(* Logix 5000 project; controller NSutherlandCapstone Emulate 5570 rev 32.11; software revision 32.00 *)

TASK MainTask (continuous, watchdog 500 ms) : MainProgram, _3WireControl, GarageDoor

MODULES
   Local : Emulate 5570 (ICP 0, rev 32.11)
      IO_Simulator : vendor 1 type 0 code 15 (ICP 3, rev 1.1, Output RPI 5 ms)
END_MODULES

VAR_GLOBAL   (* controller tags *)
   PL_G : BOOL := 1;
   PL_R : BOOL;
   SS : BOOL;
END_VAR

PROGRAM _3WireControl   (* main routine MainRoutine *)
// PLC lab 3
VAR
   Motor : BOOL;
   NCNC_AND_00 : FBD_BOOLEAN_AND := (In1 := 1, In2 := 1, In3 := 1, In4 := 1, In5 := 1, In6 := 1, In7 := 1, In8 := 1);
   NCNC_Motor_Energize : SFC_ACTION := (Status := 16#0020_0000, PauseTimer := 1);
   NCNC_NOT_00 : FBD_BOOLEAN_NOT := (In := 1);
   NCNC_OR_00 : FBD_BOOLEAN_OR;
   NCNC_SetBit : SFC_STEP := (Status := 16#0020_0000, PauseTimer := 1);
   NCNC_SetDone : BOOL;
   NCNO_AND_00 : FBD_BOOLEAN_AND := (In1 := 1, In2 := 1, In3 := 1, In4 := 1, In5 := 1, In6 := 1, In7 := 1, In8 := 1);
   NCNO_Motor_Energize : SFC_ACTION := (Status := 16#0020_0000, PauseTimer := 1);
   NCNO_OR_00 : FBD_BOOLEAN_OR;
   NCNO_SetBit : SFC_STEP := (Status := 16#0020_0000, PauseTimer := 1);
   NCNO_SetDone : BOOL;
   NONC_AND_00 : FBD_BOOLEAN_AND := (In1 := 1, In2 := 1, In3 := 1, In4 := 1, In5 := 1, In6 := 1, In7 := 1, In8 := 1);
   NONC_Motor_Energize : SFC_ACTION := (Status := 16#0020_0000, PauseTimer := 1);
   NONC_NOT_00 : FBD_BOOLEAN_NOT := (In := 1);
   NONC_NOT_01 : FBD_BOOLEAN_NOT := (In := 1);
   NONC_OR_00 : FBD_BOOLEAN_OR;
   NONC_SetBit : SFC_STEP := (Status := 16#0020_0000, PauseTimer := 1);
   NONC_SetDone : BOOL;
   NONO_AND_00 : FBD_BOOLEAN_AND := (In1 := 1, In2 := 1, In3 := 1, In4 := 1, In5 := 1, In6 := 1, In7 := 1, In8 := 1);
   NONO_Motor_Energize : SFC_ACTION := (Status := 16#0020_0000, PauseTimer := 1);
   NONO_NOT_00 : FBD_BOOLEAN_NOT := (In := 1);
   NONO_OR_00 : FBD_BOOLEAN_OR;
   NONO_SetBit : SFC_STEP := (Status := 16#0020_0000, PauseTimer := 1);
   NONO_SetDone : BOOL;
   PB1 : BOOL := 1;   // NC PB
   PB2 : BOOL;   // NO PB
   PB3 : BOOL;   // NO PB
   PB4 : BOOL := 1;   // NC PB
END_VAR

ROUTINE FBD_1_NCNO   (* function block diagram *)
   SHEET 1
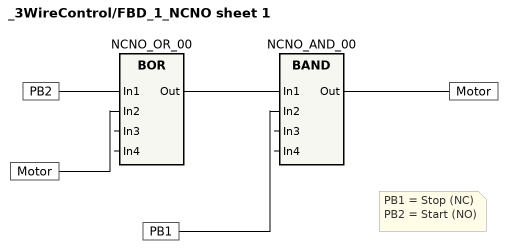
   // PB1 = Stop (NC)
   // PB2 = Start (NO)
   NCNO_OR_00 : BOR(In1 := PB2, In2 := Motor);   // unwired pins: In3 In4
   NCNO_AND_00 : BAND(In1 := NCNO_OR_00.Out, In2 := PB1);   // unwired pins: In3 In4
   Motor := NCNO_AND_00.Out;
END_ROUTINE

ROUTINE FBD_2_NONO   (* function block diagram *)
   SHEET 1
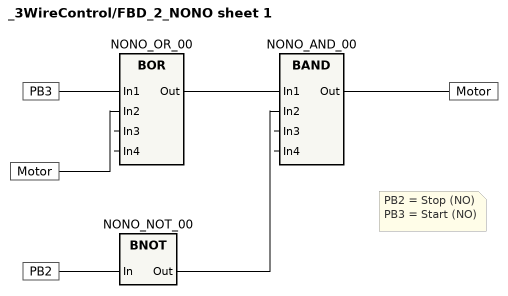
   // PB2 = Stop (NO)
   // PB3 = Start (NO)
   NONO_OR_00 : BOR(In1 := PB3, In2 := Motor);   // unwired pins: In3 In4
   NONO_NOT_00 : BNOT(In := PB2);
   NONO_AND_00 : BAND(In1 := NONO_OR_00.Out, In2 := NONO_NOT_00.Out);   // unwired pins: In3 In4
   Motor := NONO_AND_00.Out;
END_ROUTINE

ROUTINE FBD_3_NONC   (* function block diagram *)
   SHEET 1
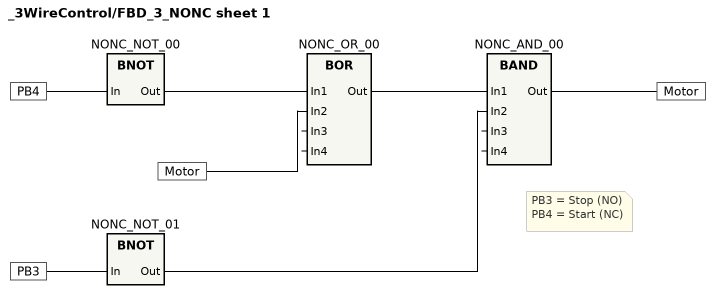
   // PB3 = Stop (NO)
   // PB4 = Start (NC)
   NONC_NOT_00 : BNOT(In := PB4);
   NONC_NOT_01 : BNOT(In := PB3);
   NONC_OR_00 : BOR(In1 := NONC_NOT_00.Out, In2 := Motor);   // unwired pins: In3 In4
   NONC_AND_00 : BAND(In1 := NONC_OR_00.Out, In2 := NONC_NOT_01.Out);   // unwired pins: In3 In4
   Motor := NONC_AND_00.Out;
END_ROUTINE

ROUTINE FBD_4_NCNC   (* function block diagram *)
   SHEET 1
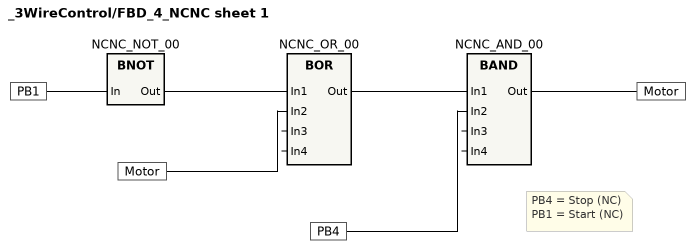
   // PB4 = Stop (NC)
   // PB1 = Start (NC)
   NCNC_NOT_00 : BNOT(In := PB1);
   NCNC_OR_00 : BOR(In1 := NCNC_NOT_00.Out, In2 := Motor);   // unwired pins: In3 In4
   NCNC_AND_00 : BAND(In1 := NCNC_OR_00.Out, In2 := PB4);   // unwired pins: In3 In4
   Motor := NCNC_AND_00.Out;
END_ROUTINE

ROUTINE MainRoutine   (* structured text *)
   JSR(SFC_3_NONC);
END_ROUTINE

ROUTINE SFC_1_NCNO   (* sequential function chart *)
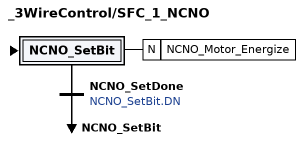
   INITIAL_STEP NCNO_SetBit:
      ACTION NCNO_Motor_Energize (N):
         Motor := PB1 & (PB2 OR Motor);
      END_ACTION
   END_STEP
   TRANSITION NCNO_SetDone FROM NCNO_SetBit TO NCNO_SetBit
      := NCNO_SetBit.DN
   END_TRANSITION
END_ROUTINE

ROUTINE SFC_2_NONO   (* sequential function chart *)
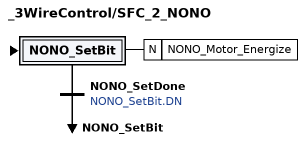
   INITIAL_STEP NONO_SetBit:
      ACTION NONO_Motor_Energize (N):
         Motor := NOT PB2 & (PB3 OR Motor);
      END_ACTION
   END_STEP
   TRANSITION NONO_SetDone FROM NONO_SetBit TO NONO_SetBit
      := NONO_SetBit.DN
   END_TRANSITION
END_ROUTINE

ROUTINE SFC_3_NONC   (* sequential function chart *)
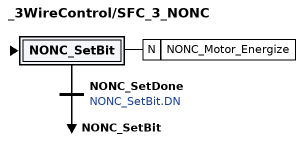
   INITIAL_STEP NONC_SetBit:
      ACTION NONC_Motor_Energize (N):
         Motor := NOT PB3 & (NOT PB4 OR Motor);
      END_ACTION
   END_STEP
   TRANSITION NONC_SetDone FROM NONC_SetBit TO NONC_SetBit
      := NONC_SetBit.DN
   END_TRANSITION
END_ROUTINE

ROUTINE SFC_4_NCNC   (* sequential function chart *)
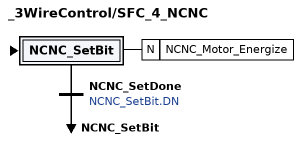
   INITIAL_STEP NCNC_SetBit:
      ACTION NCNC_Motor_Energize (N):
         Motor := PB4 & (NOT PB1 OR Motor);
      END_ACTION
   END_STEP
   TRANSITION NCNC_SetDone FROM NCNC_SetBit TO NCNC_SetBit
      := NCNC_SetBit.DN
   END_TRANSITION
END_ROUTINE

ROUTINE ST_1_NCNO   (* structured text *)
// Routine 1 of PLC lab 3
   // Lab 3 R1_NCNO
   (*
       PB1 = NC PB
       PB2 = NO PB
   *)
   
   Motor := PB1 & (PB2 OR Motor);
END_ROUTINE

ROUTINE ST_2_NONO   (* structured text *)
// Routine 2 of PLC lab 3
   // Lab 3 R2_NONO
   (*
       PB3 = NO PB
       PB2 = NO PB
   *)
   
   Motor := NOT PB2 & (PB3 OR Motor);
END_ROUTINE

ROUTINE ST_3_NONC   (* structured text *)
// Routine 3 of PLC lab 3
   // Lab 3 R3_NONC
   (*
       PB3 = NO PB
       PB4 = NC PB
   *)
   
   Motor := NOT PB3 & (NOT PB4 OR Motor);
END_ROUTINE

ROUTINE ST_4_NCNC   (* structured text *)
// Routine 4 of PLC lab 3
   // Lab 3 R4_NCNC
   (*
        PB4 = NC PB
        PB1 = NC PB
   *)
   
   Motor := PB4 & (NOT PB1 OR Motor);
END_ROUTINE
END_PROGRAM

PROGRAM GarageDoor   (* main routine MainRoutine *)
// PLC lab 4
VAR
   Ajar_LT : BOOL := 1;
   Bottom_Sensor : BOOL;
   Closed_LT : BOOL;
   Down_PB : BOOL;
   Fault_LT : BOOL;
   Halt : BOOL;
   Motor_Down : BOOL;
   Motor_Stopped : BOOL := 1;
   Motor_Up : BOOL;
   Open_LT : BOOL;
   Stop_PB : BOOL;
   Top_Sensor : BOOL;
   Up_PB : BOOL;
   Ver1_AND_00 : FBD_BOOLEAN_AND := (In1 := 1, In2 := 1, In3 := 1, In4 := 1, In5 := 1, In6 := 1, In7 := 1, In8 := 1);
   Ver1_AND_01 : FBD_BOOLEAN_AND := (In1 := 1, In2 := 1, In3 := 1, In4 := 1, In5 := 1, In6 := 1, In7 := 1, In8 := 1);
   Ver1_AND_02 : FBD_BOOLEAN_AND := (In1 := 1, In2 := 1, In3 := 1, In4 := 1, In5 := 1, In6 := 1, In7 := 1, In8 := 1);
   Ver1_AND_03 : FBD_BOOLEAN_AND := (In1 := 1, In2 := 1, In3 := 1, In4 := 1, In5 := 1, In6 := 1, In7 := 1, In8 := 1);
   Ver1_AND_04 : FBD_BOOLEAN_AND := (In1 := 1, In2 := 1, In3 := 1, In4 := 1, In5 := 1, In6 := 1, In7 := 1, In8 := 1);
   Ver1_AND_05 : FBD_BOOLEAN_AND := (In1 := 1, In2 := 1, In3 := 1, In4 := 1, In5 := 1, In6 := 1, In7 := 1, In8 := 1);
   Ver1_AND_06 : FBD_BOOLEAN_AND := (In1 := 1, In2 := 1, In3 := 1, In4 := 1, In5 := 1, In6 := 1, In7 := 1, In8 := 1);
   Ver1_AND_07 : FBD_BOOLEAN_AND := (In1 := 1, In2 := 1, In3 := 1, In4 := 1, In5 := 1, In6 := 1, In7 := 1, In8 := 1);
   Ver1_AND_08 : FBD_BOOLEAN_AND := (In1 := 1, In2 := 1, In3 := 1, In4 := 1, In5 := 1, In6 := 1, In7 := 1, In8 := 1);
   Ver1_MotorEnergize : SFC_ACTION := (Status := 16#0020_0000, PauseTimer := 1);
   Ver1_NOT_00 : FBD_BOOLEAN_NOT := (In := 1);
   Ver1_NOT_01 : FBD_BOOLEAN_NOT := (In := 1);
   Ver1_NOT_02 : FBD_BOOLEAN_NOT := (In := 1);
   Ver1_NOT_03 : FBD_BOOLEAN_NOT := (In := 1);
   Ver1_NOT_04 : FBD_BOOLEAN_NOT := (In := 1);
   Ver1_NOT_05 : FBD_BOOLEAN_NOT := (In := 1);
   Ver1_NOT_06 : FBD_BOOLEAN_NOT := (In := 1);
   Ver1_NOT_07 : FBD_BOOLEAN_NOT := (In := 1);
   Ver1_NOT_08 : FBD_BOOLEAN_NOT := (In := 1);
   Ver1_NOT_09 : FBD_BOOLEAN_NOT := (In := 1);
   Ver1_NOT_10 : FBD_BOOLEAN_NOT := (In := 1);
   Ver1_NOT_11 : FBD_BOOLEAN_NOT := (In := 1);
   Ver1_NOT_12 : FBD_BOOLEAN_NOT := (In := 1);
   Ver1_NOT_13 : FBD_BOOLEAN_NOT := (In := 1);
   Ver1_OR_00 : FBD_BOOLEAN_OR;
   Ver1_OR_01 : FBD_BOOLEAN_OR;
   Ver1_SetBit : SFC_STEP := (Status := 16#0020_0000, PauseTimer := 1);
   Ver1_SetDone : BOOL;
   Ver1_SetIndicators : SFC_ACTION := (Status := 16#0020_0000, PauseTimer := 1);
   Ver2_AND_00 : FBD_BOOLEAN_AND := (In1 := 1, In2 := 1, In3 := 1, In4 := 1, In5 := 1, In6 := 1, In7 := 1, In8 := 1);
   Ver2_AND_01 : FBD_BOOLEAN_AND := (In1 := 1, In2 := 1, In3 := 1, In4 := 1, In5 := 1, In6 := 1, In7 := 1, In8 := 1);
   Ver2_AND_02 : FBD_BOOLEAN_AND := (In1 := 1, In2 := 1, In3 := 1, In4 := 1, In5 := 1, In6 := 1, In7 := 1, In8 := 1);
   Ver2_AND_03 : FBD_BOOLEAN_AND := (In1 := 1, In2 := 1, In3 := 1, In4 := 1, In5 := 1, In6 := 1, In7 := 1, In8 := 1);
   Ver2_AND_04 : FBD_BOOLEAN_AND := (In1 := 1, In2 := 1, In3 := 1, In4 := 1, In5 := 1, In6 := 1, In7 := 1, In8 := 1);
   Ver2_AND_05 : FBD_BOOLEAN_AND := (In1 := 1, In2 := 1, In3 := 1, In4 := 1, In5 := 1, In6 := 1, In7 := 1, In8 := 1);
   Ver2_AND_06 : FBD_BOOLEAN_AND := (In1 := 1, In2 := 1, In3 := 1, In4 := 1, In5 := 1, In6 := 1, In7 := 1, In8 := 1);
   Ver2_AND_07 : FBD_BOOLEAN_AND := (In1 := 1, In2 := 1, In3 := 1, In4 := 1, In5 := 1, In6 := 1, In7 := 1, In8 := 1);
   Ver2_AND_08 : FBD_BOOLEAN_AND := (In1 := 1, In2 := 1, In3 := 1, In4 := 1, In5 := 1, In6 := 1, In7 := 1, In8 := 1);
   Ver2_AND_09 : FBD_BOOLEAN_AND := (In1 := 1, In2 := 1, In3 := 1, In4 := 1, In5 := 1, In6 := 1, In7 := 1, In8 := 1);
   Ver2_AND_10 : FBD_BOOLEAN_AND := (In1 := 1, In2 := 1, In3 := 1, In4 := 1, In5 := 1, In6 := 1, In7 := 1, In8 := 1);
   Ver2_AND_11 : FBD_BOOLEAN_AND := (In1 := 1, In2 := 1, In3 := 1, In4 := 1, In5 := 1, In6 := 1, In7 := 1, In8 := 1);
   Ver2_AND_12 : FBD_BOOLEAN_AND := (In1 := 1, In2 := 1, In3 := 1, In4 := 1, In5 := 1, In6 := 1, In7 := 1, In8 := 1);
   Ver2_CheckAjar : BOOL;
   Ver2_CheckClosed : BOOL;
   Ver2_CheckDown : BOOL;
   Ver2_CheckFault : BOOL;
   Ver2_CheckHalt : BOOL;
   Ver2_CheckOpen : BOOL;
   Ver2_CheckStopped : BOOL;
   Ver2_CheckUp : BOOL;
   Ver2_DoneAjar : BOOL;
   Ver2_DoneClosed : BOOL;
   Ver2_DoneDown : BOOL;
   Ver2_DoneFault : BOOL;
   Ver2_DoneHalt : BOOL;
   Ver2_DoneOpen : BOOL;
   Ver2_DoneStopped : BOOL;
   Ver2_DoneUp : BOOL;
   Ver2_MotorEnergize : SFC_ACTION := (Status := 16#0020_0000, PauseTimer := 1);
   Ver2_NOT_00 : FBD_BOOLEAN_NOT := (In := 1);
   Ver2_NOT_01 : FBD_BOOLEAN_NOT := (In := 1);
   Ver2_NOT_02 : FBD_BOOLEAN_NOT := (In := 1);
   Ver2_NOT_03 : FBD_BOOLEAN_NOT := (In := 1);
   Ver2_NOT_04 : FBD_BOOLEAN_NOT := (In := 1);
   Ver2_NOT_05 : FBD_BOOLEAN_NOT := (In := 1);
   Ver2_NOT_06 : FBD_BOOLEAN_NOT := (In := 1);
   Ver2_NOT_07 : FBD_BOOLEAN_NOT := (In := 1);
   Ver2_NOT_08 : FBD_BOOLEAN_NOT := (In := 1);
   Ver2_NOT_09 : FBD_BOOLEAN_NOT := (In := 1);
   Ver2_NOT_10 : FBD_BOOLEAN_NOT := (In := 1);
   Ver2_NOT_11 : FBD_BOOLEAN_NOT := (In := 1);
   Ver2_NOT_12 : FBD_BOOLEAN_NOT := (In := 1);
   Ver2_NOT_13 : FBD_BOOLEAN_NOT := (In := 1);
   Ver2_OR_00 : FBD_BOOLEAN_OR;
   Ver2_OR_01 : FBD_BOOLEAN_OR;
   Ver2_OR_02 : FBD_BOOLEAN_OR;
   Ver2_OR_03 : FBD_BOOLEAN_OR;
   Ver2_OR_04 : FBD_BOOLEAN_OR;
   Ver2_SetAjar : SFC_ACTION := (Status := 16#0020_0000, PauseTimer := 1);
   Ver2_SetBit : SFC_STEP := (Status := 16#0020_0000, PauseTimer := 1);
   Ver2_SetBit0 : SFC_STEP := (Status := 16#0020_0000, PauseTimer := 1);
   Ver2_SetBit1 : SFC_STEP := (Status := 16#0020_0000, PauseTimer := 1);
   Ver2_SetBit2 : SFC_STEP := (Status := 16#0020_0000, PauseTimer := 1);
   Ver2_SetBit3 : SFC_STEP := (Status := 16#0020_0000, PauseTimer := 1);
   Ver2_SetBit4 : SFC_STEP := (Status := 16#0020_0000, PauseTimer := 1);
   Ver2_SetBit5 : SFC_STEP := (Status := 16#0020_0000, PauseTimer := 1);
   Ver2_SetBit6 : SFC_STEP := (Status := 16#0020_0000, PauseTimer := 1);
   Ver2_SetBit7 : SFC_STEP := (Status := 16#0020_0000, PauseTimer := 1);
   Ver2_SetClosed : SFC_ACTION := (Status := 16#0020_0000, PauseTimer := 1);
   Ver2_SetDone : BOOL;
   Ver2_SetDown : SFC_ACTION := (Status := 16#0020_0000, PauseTimer := 1);
   Ver2_SetFault : SFC_ACTION := (Status := 16#0020_0000, PauseTimer := 1);
   Ver2_SetHalt : SFC_ACTION := (Status := 16#0020_0000, PauseTimer := 1);
   Ver2_SetIndicators : SFC_ACTION := (Status := 16#0020_0000, PauseTimer := 1);
   Ver2_SetOpen : SFC_ACTION := (Status := 16#0020_0000, PauseTimer := 1);
   Ver2_SetStopped : SFC_ACTION := (Status := 16#0020_0000, PauseTimer := 1);
   Ver2_SetUp : SFC_ACTION := (Status := 16#0020_0000, PauseTimer := 1);
   Ver2_Start : SFC_STEP := (Status := 16#0020_0000, PauseTimer := 1);
END_VAR

ROUTINE FBD_Ver1   (* function block diagram *)
   SHEET 1   // Motor Up
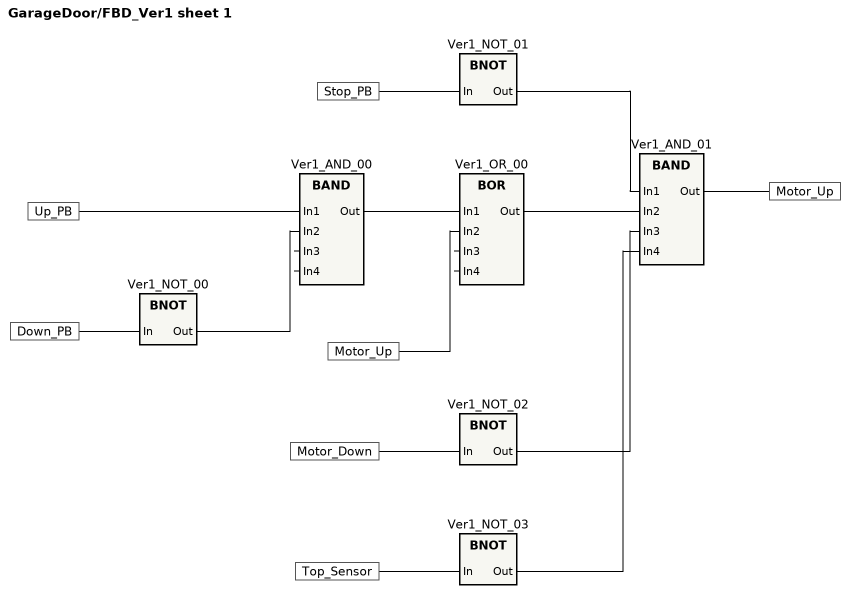
   Ver1_NOT_00 : BNOT(In := Down_PB);
   Ver1_AND_00 : BAND(In1 := Up_PB, In2 := Ver1_NOT_00.Out);   // unwired pins: In3 In4
   Ver1_NOT_01 : BNOT(In := Stop_PB);
   Ver1_OR_00 : BOR(In1 := Ver1_AND_00.Out, In2 := Motor_Up);   // unwired pins: In3 In4
   Ver1_NOT_02 : BNOT(In := Motor_Down);
   Ver1_NOT_03 : BNOT(In := Top_Sensor);
   Ver1_AND_01 : BAND(In1 := Ver1_NOT_01.Out, In2 := Ver1_OR_00.Out, In3 := Ver1_NOT_02.Out, In4 := Ver1_NOT_03.Out);
   Motor_Up := Ver1_AND_01.Out;
   SHEET 2   // Motor Down
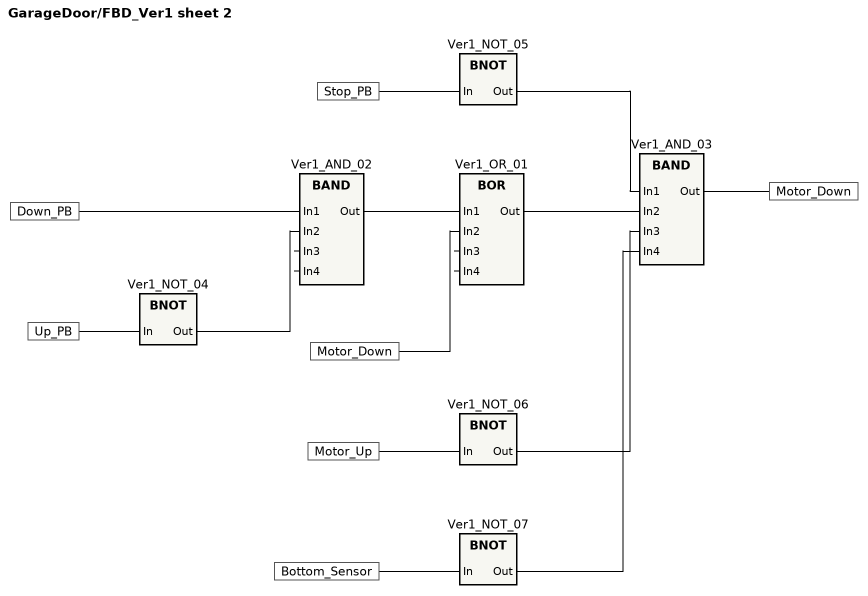
   Ver1_NOT_04 : BNOT(In := Up_PB);
   Ver1_AND_02 : BAND(In1 := Down_PB, In2 := Ver1_NOT_04.Out);   // unwired pins: In3 In4
   Ver1_NOT_05 : BNOT(In := Stop_PB);
   Ver1_OR_01 : BOR(In1 := Ver1_AND_02.Out, In2 := Motor_Down);   // unwired pins: In3 In4
   Ver1_NOT_06 : BNOT(In := Motor_Up);
   Ver1_NOT_07 : BNOT(In := Bottom_Sensor);
   Ver1_AND_03 : BAND(In1 := Ver1_NOT_05.Out, In2 := Ver1_OR_01.Out, In3 := Ver1_NOT_06.Out, In4 := Ver1_NOT_07.Out);
   Motor_Down := Ver1_AND_03.Out;
   SHEET 3   // Signals
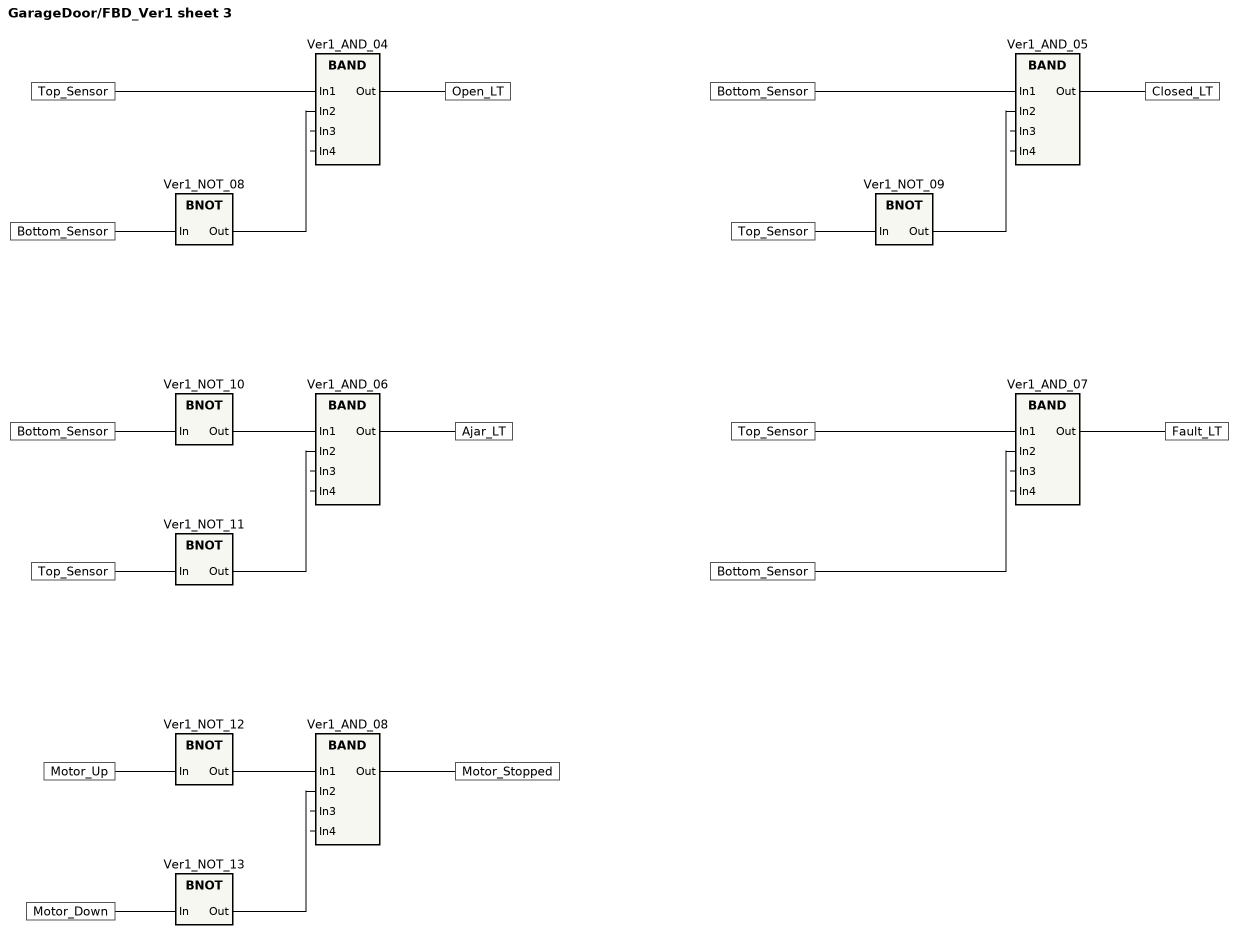
   Ver1_NOT_08 : BNOT(In := Bottom_Sensor);
   Ver1_NOT_10 : BNOT(In := Bottom_Sensor);
   Ver1_NOT_11 : BNOT(In := Top_Sensor);
   Ver1_NOT_12 : BNOT(In := Motor_Up);
   Ver1_NOT_13 : BNOT(In := Motor_Down);
   Ver1_AND_04 : BAND(In1 := Top_Sensor, In2 := Ver1_NOT_08.Out);   // unwired pins: In3 In4
   Ver1_AND_06 : BAND(In1 := Ver1_NOT_10.Out, In2 := Ver1_NOT_11.Out);   // unwired pins: In3 In4
   Ver1_AND_08 : BAND(In1 := Ver1_NOT_12.Out, In2 := Ver1_NOT_13.Out);   // unwired pins: In3 In4
   Open_LT := Ver1_AND_04.Out;
   Ajar_LT := Ver1_AND_06.Out;
   Motor_Stopped := Ver1_AND_08.Out;
   Ver1_NOT_09 : BNOT(In := Top_Sensor);
   Ver1_AND_05 : BAND(In1 := Bottom_Sensor, In2 := Ver1_NOT_09.Out);   // unwired pins: In3 In4
   Ver1_AND_07 : BAND(In1 := Top_Sensor, In2 := Bottom_Sensor);   // unwired pins: In3 In4
   Closed_LT := Ver1_AND_05.Out;
   Fault_LT := Ver1_AND_07.Out;
END_ROUTINE

ROUTINE FBD_Ver2   (* function block diagram *)
   SHEET 1   // Motor Up
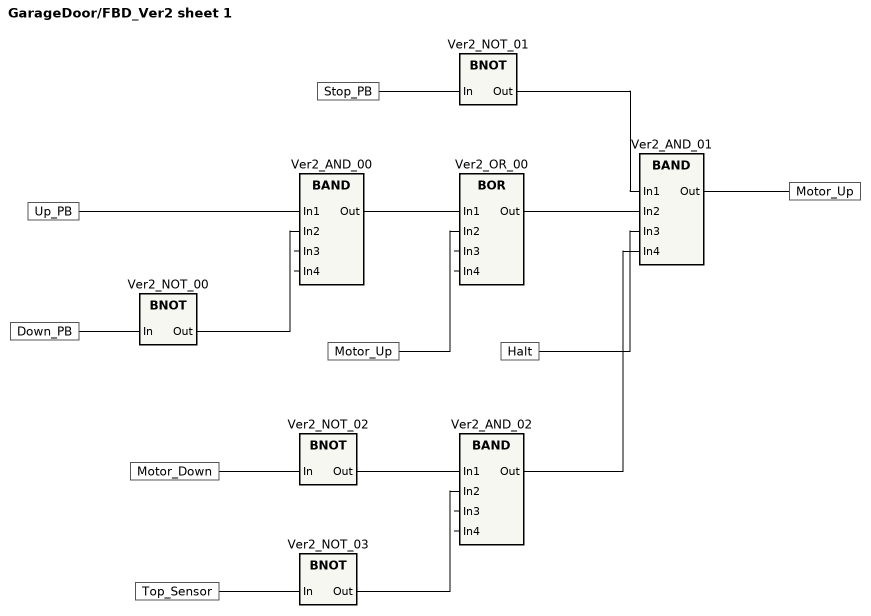
   Ver2_NOT_00 : BNOT(In := Down_PB);
   Ver2_AND_00 : BAND(In1 := Up_PB, In2 := Ver2_NOT_00.Out);   // unwired pins: In3 In4
   Ver2_NOT_02 : BNOT(In := Motor_Down);
   Ver2_NOT_03 : BNOT(In := Top_Sensor);
   Ver2_NOT_01 : BNOT(In := Stop_PB);
   Ver2_OR_00 : BOR(In1 := Ver2_AND_00.Out, In2 := Motor_Up);   // unwired pins: In3 In4
   Ver2_AND_02 : BAND(In1 := Ver2_NOT_02.Out, In2 := Ver2_NOT_03.Out);   // unwired pins: In3 In4
   Ver2_AND_01 : BAND(In1 := Ver2_NOT_01.Out, In2 := Ver2_OR_00.Out, In3 := Halt, In4 := Ver2_AND_02.Out);
   Motor_Up := Ver2_AND_01.Out;
   SHEET 2   // Motor Down
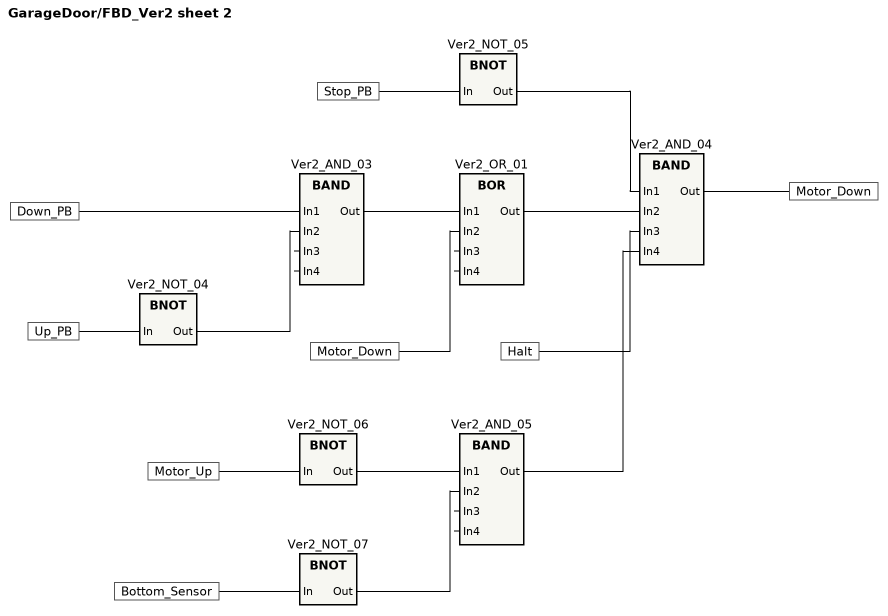
   Ver2_NOT_04 : BNOT(In := Up_PB);
   Ver2_AND_03 : BAND(In1 := Down_PB, In2 := Ver2_NOT_04.Out);   // unwired pins: In3 In4
   Ver2_NOT_06 : BNOT(In := Motor_Up);
   Ver2_NOT_07 : BNOT(In := Bottom_Sensor);
   Ver2_NOT_05 : BNOT(In := Stop_PB);
   Ver2_OR_01 : BOR(In1 := Ver2_AND_03.Out, In2 := Motor_Down);   // unwired pins: In3 In4
   Ver2_AND_05 : BAND(In1 := Ver2_NOT_06.Out, In2 := Ver2_NOT_07.Out);   // unwired pins: In3 In4
   Ver2_AND_04 : BAND(In1 := Ver2_NOT_05.Out, In2 := Ver2_OR_01.Out, In3 := Halt, In4 := Ver2_AND_05.Out);
   Motor_Down := Ver2_AND_04.Out;
   SHEET 3   // Signals
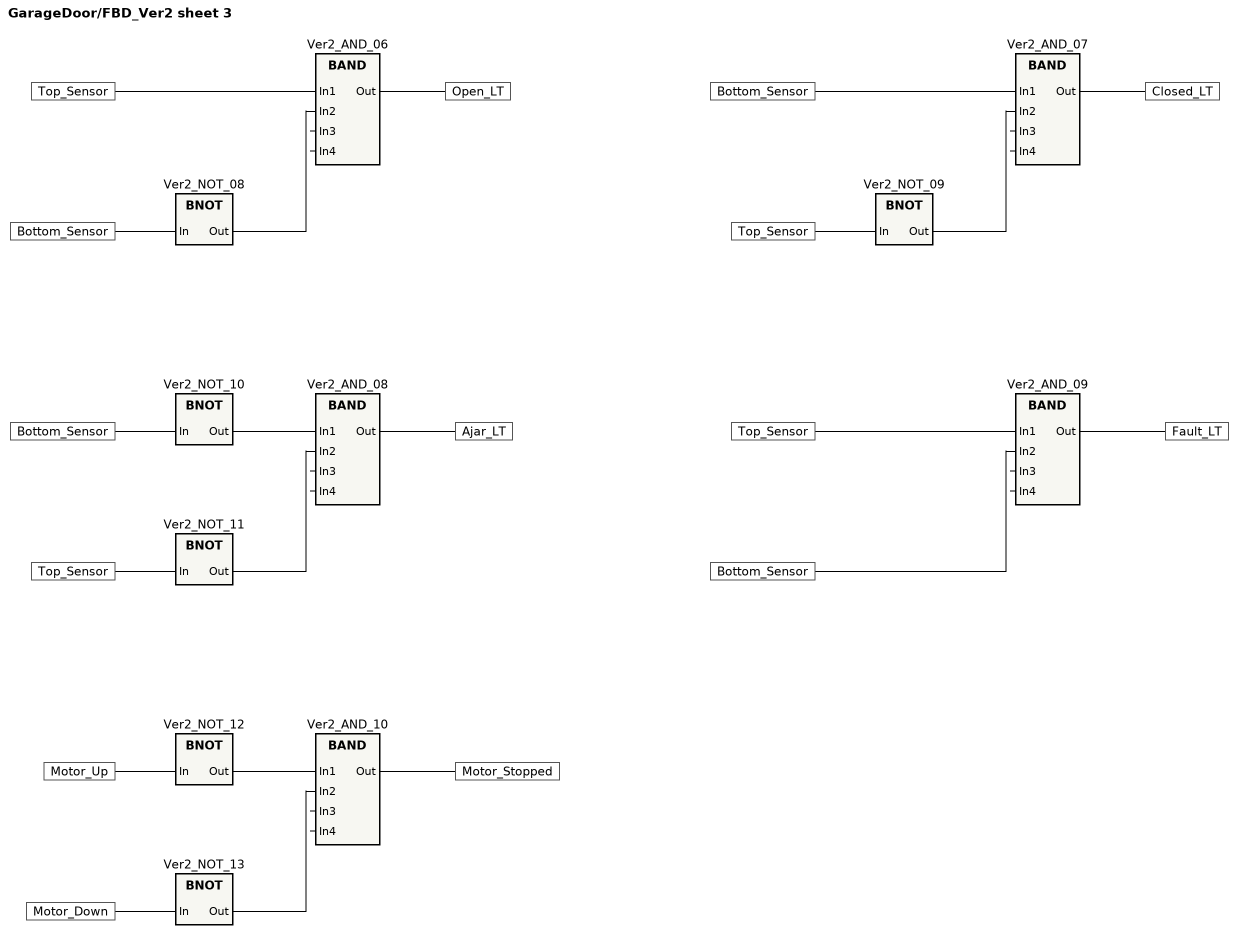
   Ver2_NOT_08 : BNOT(In := Bottom_Sensor);
   Ver2_NOT_10 : BNOT(In := Bottom_Sensor);
   Ver2_NOT_11 : BNOT(In := Top_Sensor);
   Ver2_NOT_12 : BNOT(In := Motor_Up);
   Ver2_NOT_13 : BNOT(In := Motor_Down);
   Ver2_AND_06 : BAND(In1 := Top_Sensor, In2 := Ver2_NOT_08.Out);   // unwired pins: In3 In4
   Ver2_AND_08 : BAND(In1 := Ver2_NOT_10.Out, In2 := Ver2_NOT_11.Out);   // unwired pins: In3 In4
   Ver2_AND_10 : BAND(In1 := Ver2_NOT_12.Out, In2 := Ver2_NOT_13.Out);   // unwired pins: In3 In4
   Open_LT := Ver2_AND_06.Out;
   Ajar_LT := Ver2_AND_08.Out;
   Motor_Stopped := Ver2_AND_10.Out;
   Ver2_NOT_09 : BNOT(In := Top_Sensor);
   Ver2_AND_07 : BAND(In1 := Bottom_Sensor, In2 := Ver2_NOT_09.Out);   // unwired pins: In3 In4
   Ver2_AND_09 : BAND(In1 := Top_Sensor, In2 := Bottom_Sensor);   // unwired pins: In3 In4
   Closed_LT := Ver2_AND_07.Out;
   Fault_LT := Ver2_AND_09.Out;
   SHEET 4   // Halt
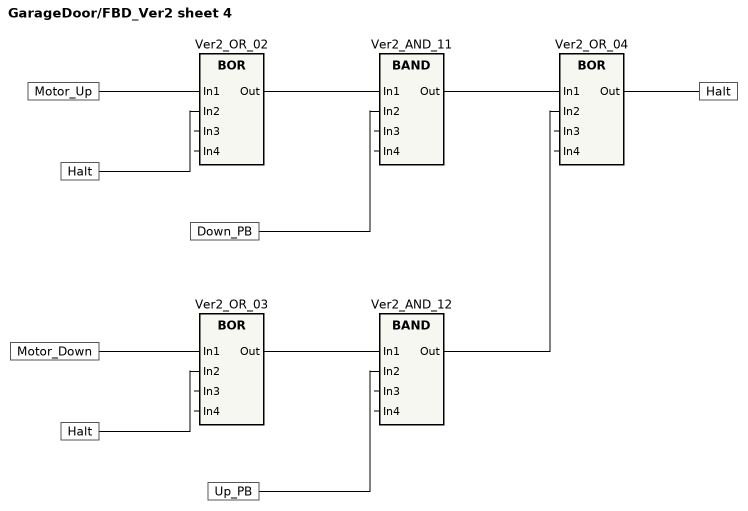
   Ver2_OR_02 : BOR(In1 := Motor_Up, In2 := Halt);   // unwired pins: In3 In4
   Ver2_OR_03 : BOR(In1 := Motor_Down, In2 := Halt);   // unwired pins: In3 In4
   Ver2_AND_11 : BAND(In1 := Ver2_OR_02.Out, In2 := Down_PB);   // unwired pins: In3 In4
   Ver2_AND_12 : BAND(In1 := Ver2_OR_03.Out, In2 := Up_PB);   // unwired pins: In3 In4
   Ver2_OR_04 : BOR(In1 := Ver2_AND_11.Out, In2 := Ver2_AND_12.Out);   // unwired pins: In3 In4
   Halt := Ver2_OR_04.Out;
END_ROUTINE

ROUTINE MainRoutine   (* structured text *)
   JSR(SFC_Ver2);
END_ROUTINE

ROUTINE SFC_Ver1   (* sequential function chart *)
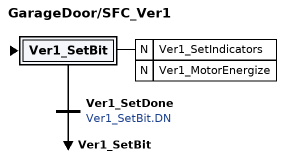
   INITIAL_STEP Ver1_SetBit:
      ACTION Ver1_SetIndicators (N):
         Open_LT       := Top_Sensor     & NOT Bottom_Sensor;
         Closed_LT     := NOT Top_Sensor & Bottom_Sensor;
         Ajar_LT       := NOT Top_Sensor & NOT Bottom_Sensor;
         Fault_LT      := Top_Sensor     & Bottom_Sensor;
         Motor_Stopped := NOT Motor_Up   & NOT Motor_Down;
      END_ACTION
      ACTION Ver1_MotorEnergize (N):
         Motor_Up   := NOT Stop_PB &
         			  ((Up_PB & NOT Down_PB) OR Motor_Up) &
         			  NOT Motor_Down &
         			  NOT Top_Sensor;
         
         Motor_Down := NOT Stop_PB &
         			  ((Down_PB & NOT Up_PB) OR Motor_Down) &
         			  NOT Motor_Up &
         			  NOT Bottom_Sensor;
      END_ACTION
   END_STEP
   TRANSITION Ver1_SetDone FROM Ver1_SetBit TO Ver1_SetBit
      := Ver1_SetBit.DN
   END_TRANSITION
END_ROUTINE

ROUTINE SFC_Ver2   (* sequential function chart *)
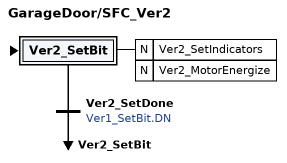
   INITIAL_STEP Ver2_SetBit:
      ACTION Ver2_SetIndicators (N):
         Open_LT       := Top_Sensor     & NOT Bottom_Sensor;
         Closed_LT     := NOT Top_Sensor & Bottom_Sensor;
         Ajar_LT       := NOT Top_Sensor & NOT Bottom_Sensor;
         Fault_LT      := Top_Sensor     & Bottom_Sensor;
         Motor_Stopped := NOT Motor_Up   & NOT Motor_Down;
         Halt		  := ((Motor_Up OR Halt) & Down_PB) OR
         				 ((Motor_Down OR Halt) & Up_PB);
      END_ACTION
      ACTION Ver2_MotorEnergize (N):
         Motor_Up      := NOT Stop_PB &
         				 NOT Halt &
                          ((Up_PB & NOT Down_PB) OR Motor_Up) &
                          NOT Motor_Down &
                          NOT Top_Sensor;
         
         Motor_Down    := NOT Stop_PB &
         				 NOT Halt &
                          ((Down_PB & NOT Up_PB) OR Motor_Down) &
                          NOT Motor_Up &
                          NOT Bottom_Sensor;
      END_ACTION
   END_STEP
   TRANSITION Ver2_SetDone FROM Ver2_SetBit TO Ver2_SetBit
      := Ver1_SetBit.DN
   END_TRANSITION
END_ROUTINE

ROUTINE ST_Ver1   (* structured text *)
   // Lab 4 Garage Door
   (*
       Version 1
       Each PB has a single function
   *)
   
   Open_LT       := Top_Sensor     & NOT Bottom_Sensor;
   Closed_LT     := NOT Top_Sensor & Bottom_Sensor;
   Ajar_LT       := NOT Top_Sensor & NOT Bottom_Sensor;
   Fault_LT      := Top_Sensor     & Bottom_Sensor;
   Motor_Stopped := NOT Motor_Up   & NOT Motor_Down;
   
   Motor_Up      := NOT Stop_PB &
                    ((Up_PB & NOT Down_PB) OR Motor_Up) &
                    NOT Motor_Down &
                    NOT Top_Sensor;
   
   Motor_Down    := NOT Stop_PB &
                    ((Down_PB & NOT Up_PB) OR Motor_Down) &
                    NOT Motor_Up &
                    NOT Bottom_Sensor;
END_ROUTINE

ROUTINE ST_Ver2   (* structured text *)
   // Lab 4 Garage Door
   (*
       Version 2
       UP & DOWN buttons also serve as STOP buttons
   	(Motor will not change direction without stopping first)
   *)
   
   Open_LT       := Top_Sensor     & NOT Bottom_Sensor;
   Closed_LT     := NOT Top_Sensor & Bottom_Sensor;
   Ajar_LT       := NOT Top_Sensor & NOT Bottom_Sensor;
   Fault_LT      := Top_Sensor     & Bottom_Sensor;
   Motor_Stopped := NOT Motor_Up   & NOT Motor_Down;
   Halt		  := ((Motor_Up OR Halt) & Down_PB) OR
   				 ((Motor_Down OR Halt) & Up_PB);
   
   Motor_Up      := NOT Stop_PB &
   				 NOT Halt &
                    ((Up_PB & NOT Down_PB) OR Motor_Up) &
                    NOT Motor_Down &
                    NOT Top_Sensor;
   
   Motor_Down    := NOT Stop_PB &
   				 NOT Halt &
                    ((Down_PB & NOT Up_PB) OR Motor_Down) &
                    NOT Motor_Up &
                    NOT Bottom_Sensor;
END_ROUTINE
END_PROGRAM

PROGRAM MainProgram   (* main routine MainRoutine *)
VAR
   A : BOOL := 1;
   AndOr_AND_00 : FBD_BOOLEAN_AND := (In1 := 1, In2 := 1, In3 := 1, In4 := 1, In5 := 1, In6 := 1, In7 := 1, In8 := 1);
   AndOr_AND_01 : FBD_BOOLEAN_AND := (In1 := 1, In2 := 1, In3 := 1, In4 := 1, In5 := 1, In6 := 1, In7 := 1, In8 := 1);
   AndOr_AND_02 : FBD_BOOLEAN_AND := (In1 := 1, In2 := 1, In3 := 1, In4 := 1, In5 := 1, In6 := 1, In7 := 1, In8 := 1);
   AndOr_AND_03 : FBD_BOOLEAN_AND := (In1 := 1, In2 := 1, In3 := 1, In4 := 1, In5 := 1, In6 := 1, In7 := 1, In8 := 1);
   AndOr_AND_04 : FBD_BOOLEAN_AND := (In1 := 1, In2 := 1, In3 := 1, In4 := 1, In5 := 1, In6 := 1, In7 := 1, In8 := 1);
   AndOr_NOT_00 : FBD_BOOLEAN_NOT := (In := 1);
   AndOr_NOT_01 : FBD_BOOLEAN_NOT := (In := 1);
   AndOr_NOT_02 : FBD_BOOLEAN_NOT := (In := 1);
   AndOr_NOT_03 : FBD_BOOLEAN_NOT := (In := 1);
   AndOr_NOT_04 : FBD_BOOLEAN_NOT := (In := 1);
   AndOr_OR_00 : FBD_BOOLEAN_OR;
   AndOr_OR_01 : FBD_BOOLEAN_OR;
   AndOr_SetBit : SFC_STEP := (Status := 16#0020_0000, PauseTimer := 1);
   AndOr_SetDone : BOOL;
   AndOr_SetPL1 : SFC_ACTION := (Status := 16#0020_0000, PauseTimer := 1);
   AndOr_SetPL2 : SFC_ACTION := (Status := 16#0020_0000, PauseTimer := 1);
   AndOr_SetPL3 : SFC_ACTION := (Status := 16#0020_0000, PauseTimer := 1);
   AndOr_SetPL4 : SFC_ACTION := (Status := 16#0020_0000, PauseTimer := 1);
   B : BOOL;
   C : BOOL := 1;
   CARRY_OUT : BOOL := 1;
   FullAdder_AND_00 : FBD_BOOLEAN_AND := (In1 := 1, In2 := 1, In3 := 1, In4 := 1, In5 := 1, In6 := 1, In7 := 1, In8 := 1);
   FullAdder_AND_01 : FBD_BOOLEAN_AND := (In1 := 1, In2 := 1, In3 := 1, In4 := 1, In5 := 1, In6 := 1, In7 := 1, In8 := 1);
   FullAdder_OR_00 : FBD_BOOLEAN_OR;
   FullAdder_SetBit : SFC_STEP := (Status := 16#0020_0000, PauseTimer := 1);
   FullAdder_SetCarry : SFC_ACTION := (Status := 16#0020_0000, PauseTimer := 1);
   FullAdder_SetDone : BOOL;
   FullAdder_SetSum : SFC_ACTION := (Status := 16#0020_0000, PauseTimer := 1);
   FullAdder_XOR_00 : FBD_BOOLEAN_XOR;
   FullAdder_XOR_01 : FBD_BOOLEAN_XOR;
   OutputNOR : BOOL := 1;
   OutputXOR : BOOL;
   PB1 : BOOL;   // NO PB
   PB2 : BOOL := 1;   // NC PB
   PB3 : BOOL := 1;   // NC PB
   PB4 : BOOL;   // NO PB
   PL1 : BOOL;
   PL2 : BOOL;
   PL3 : BOOL;
   PL4 : BOOL;
   SUM_OUT : BOOL;
   TruthTables_NOT_00 : FBD_BOOLEAN_NOT := (In := 1);
   TruthTables_NOT_01 : FBD_BOOLEAN_NOT := (In := 1);
   TruthTables_OR_00 : FBD_BOOLEAN_OR;
   TruthTables_SetBit : SFC_STEP := (Status := 16#0020_0000, PauseTimer := 1);
   TruthTables_SetDone : BOOL;
   TruthTables_SetNOR : SFC_ACTION := (Status := 16#0020_0000, PauseTimer := 1);
   TruthTables_SetXOR : SFC_ACTION := (Status := 16#0020_0000, PauseTimer := 1);
   TruthTables_XOR_00 : FBD_BOOLEAN_XOR;
   XICXIO_NOT_00 : FBD_BOOLEAN_NOT := (Out := 1);
   XICXIO_NOT_01 : FBD_BOOLEAN_NOT := (Out := 1);
   XICXIO_SetBit : SFC_STEP := (Status := 16#0020_0000, PauseTimer := 1);
   XICXIO_SetDone : BOOL;
   XICXIO_SetPL1 : SFC_ACTION := (Status := 16#0020_0000, PauseTimer := 1);
   XICXIO_SetPL2 : SFC_ACTION := (Status := 16#0020_0000, PauseTimer := 1);
   XICXIO_SetPL3 : SFC_ACTION := (Status := 16#0020_0000, PauseTimer := 1);
   XICXIO_SetPL4 : SFC_ACTION := (Status := 16#0020_0000, PauseTimer := 1);
END_VAR

ROUTINE FBD_1_XICXIO   (* function block diagram *)
   SHEET 1
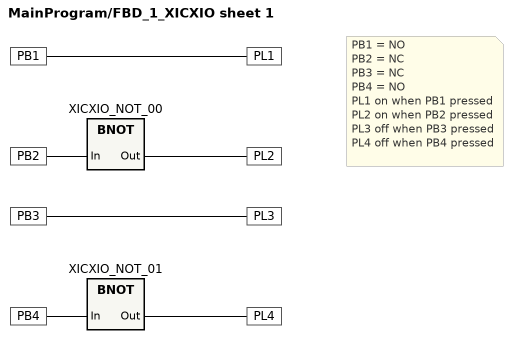
   // PB1 = NO
   // PB2 = NC
   // PB3 = NC
   // PB4 = NO
   // PL1 on when PB1 pressed
   // PL2 on when PB2 pressed
   // PL3 off when PB3 pressed
   // PL4 off when PB4 pressed
   XICXIO_NOT_00 : BNOT(In := PB2);
   XICXIO_NOT_01 : BNOT(In := PB4);
   PL1 := PB1;
   PL2 := XICXIO_NOT_00.Out;
   PL3 := PB3;
   PL4 := XICXIO_NOT_01.Out;
END_ROUTINE
